// TIA Portal V19 export
TYPE "A0302_Manager_Ctrl"
   STRUCT
      EnableStopDoorOpeningReq : Bool := TRUE;
      EnableStopInPhase : Bool := TRUE;
      EnableStopProgrammed : Bool := TRUE;
      Control_ON : Bool := FALSE;
      REST_Req : Bool;
      WORK_Req : Bool;
      Rest : Bool;
      Work : Bool;
   END_STRUCT;
END_TYPE
